Yaskawa INFORM job: MOVJ.JBI

/JOB
//NAME MOVJ
//POS
///NPOS 2,2,0,0,0,0
///TOOL 0
///POSTYPE PULSE
///PULSE
C00000=9504,-120137,-73275,91468,-72711,6858
C00001=9504,-120137,-73275,91468,-72711,6858
BC00000=379783,663794,170794
BC00001=9119,663794,170794
//INST
///DATE 2025/04/11 21:11
///ATTR SC,RW
///GROUP1 RB1,BS1
NOP
*LABEL
MOVJ C00000 BC00000 VJ=75.00
MOVJ C00001 BC00001 VJ=75.00
JUMP *LABEL
END
